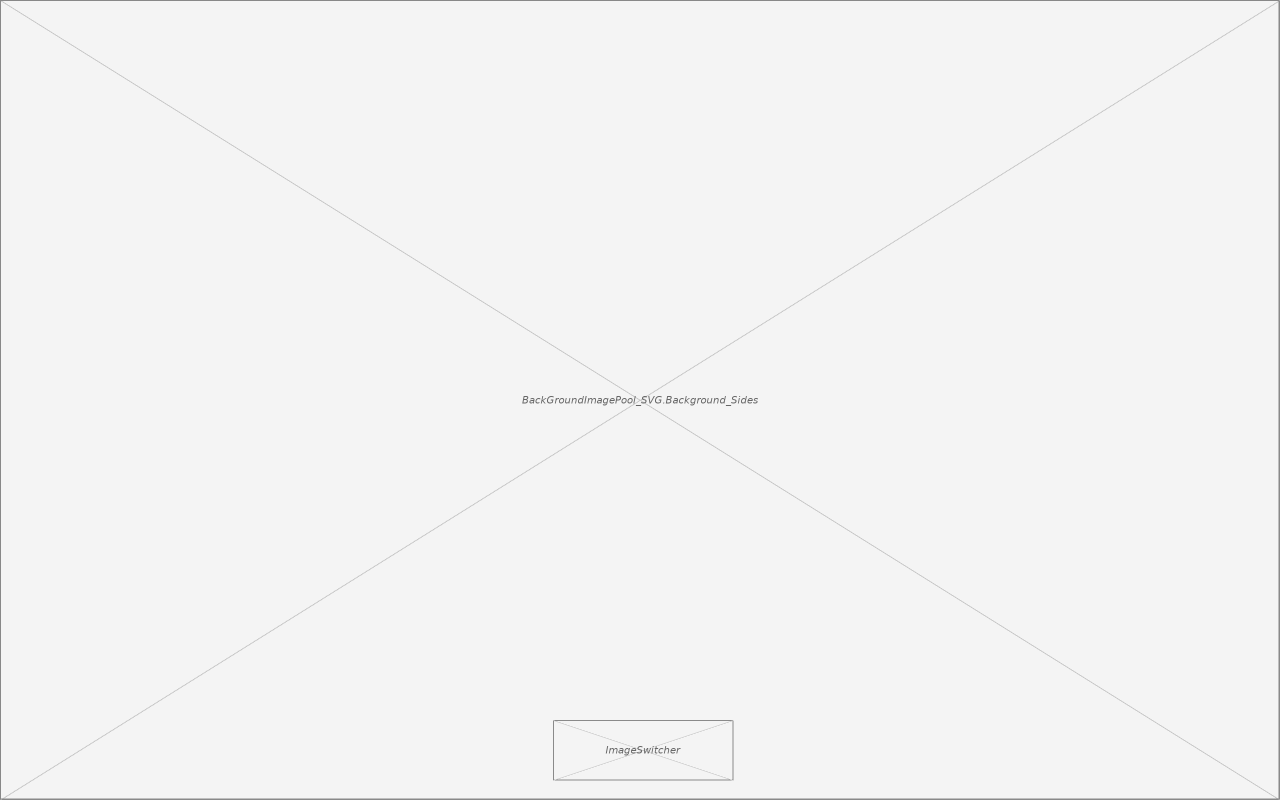
VISUALIZATION BackgroundWithBorder  // 1280x800
    Image (0,710 1280x90), image: BackGroundImagePool_SVG.Background_Bottom
    Image (0,0 1280x800), invisible if: GVL_HMI.fbHMIControl.bHideBorders, image: BackGroundImagePool_SVG.Background_Sides
    ImageSwitcher (553,720 180x60), variable: GVL_HMI.bCmdSettings, input disabled if: GVL_HMI.fbHMIControl.bDisableSettings, background image: Buttons_SVG.Home-Settings Switch Pushed, image: Buttons_SVG.Home Settings switch, behaviour: TOGGLE
        p3148411668: Buttons_SVG.Home-Settings Switch Pushed
END_VISUALIZATION

(* stored: Version 1.1.0.1, ProductVersion 3.1.4024.11
   Visu BackgroundWithBorder: Id {80a01c00-7e95-43c6-ba37-e4848c79e10a} *)
